// TIA Portal V19 export
VAR_GLOBAL   // PLC tag table "EM90_Template"
END_VAR
VAR_GLOBAL CONSTANT   // user constants
   NMAX_ERROR_NOREACTION_EM90 : Int := 1;   // Number of Error (no reaction) type alarms
   NMAX_ERROR_ABORT_EM90 : Int := 1;   // Number of Error (command abort) type alarms
   NMAX_ERROR_STOP_EM90 : Int := 50;   // Number of Error (command stop) type alarms
   NMAX_WARNING_NOREACTION_EM90 : Int := 1;   // Number of Warning (no reaction) type alarms
   NMAX_WARNING_HOLD_EM90 : Int := 1;   // Number of Warning (command hold) type alarms
   NMAX_WARNING_SUSPEND_EM90 : Int := 1;   // Number of Warning (command suspend) type alarms
   NMAX_INFORMATION_EM90 : Int := 1;   // Number of Information type alarms
   NMAX_CRITERIAANALYSIS_EM90 : Int := 1;   // Criteria analysis
END_VAR
